// TIA Portal V17 export
// export: Created 2022-06-16T09:21:05.2505257Z, ExportSetting WithDefaults, DisplayName Totally Integrated Automation Portal, DisplayVersion V17, DisplayName TIA Portal Openness, DisplayVersion V17, DisplayName TIA Portal Version Control Interface, DisplayVersion V17, DisplayName STEP 7 Professional, DisplayVersion V17, DisplayName STEP 7 Safety, DisplayVersion V17, DisplayName WinCC Advanced, DisplayVersion V17
DATA_BLOCK "DB_Params"   // DB70
{ S7_Optimized_Access := 'TRUE' }
VERSION : 0.1
// stored: AutoNumber false, DBAccessibleFromOPCUA true, IsOnlyStoredInLoadMemory false, IsRetainMemResEnabled false, IsWriteProtectedInAS false, MemoryReserve 100
   VAR
      SensorAngle : Real;   // angle absolu donné par capteur position [Rad]
      SensorAngleOffset : Real;   // Pour les capteurs 1 tour = pi / pour les capteurs 8 tours = 8*pi
      PinionModule : Real;   // Module pinion capteur pos [m] (std actuel : 3e-3)
      PinionTeethNum : Real;   // Nombre de dents du pinion (std actuel : 15)
   END_VAR
BEGIN
END_DATA_BLOCK
